// TIA Portal V19 export
DATA_BLOCK "RollformingMng"   // DB157
{ DB_Accessible_From_OPC_UA := 'FALSE' }
// stored: DBAccessibleFromOPCUA false, InstanceOfName RollformingMng_FB, InstanceOfType FB
"RollformingMng_FB"
   // VAR_INPUT
   //    AreaInterface : "AreaInterface";
   //    ZSI_Area : "udt_ZoneSafetyInterface";
   //    DataIn : Struct
   //       PbMaterialFwd : Bool;
   //       PbCutRest : Bool;
   //       PbCutWork : Bool;
   //       SensorMatPresence_Entry : Bool;
   //       SensorMatPresence_BeforeMW : Bool;
   //       SensorMatPresence_AfterMW : Bool;
   //       SensorMatPresence_ConveyorEntry : Bool;
   //    END_STRUCT;
   //    CIn : Struct
   //       PitTable : Struct
   //          IsAtRest : Bool;
   //          IsAtWork : Bool;
   //       END_STRUCT;
   //       Upstream : Struct
   //          EnableMove : Bool;
   //          InCycleOrEmptying : Bool;
   //          NextEndOfMaterial : Bool;
   //       END_STRUCT;
   //       PPrf : "PPrf_Data";
   //       ProdManager : "Prod_Part_Ctrl";
   //       Rollformer : Struct
   //          IsStandstill : Bool;
   //          InTargetPosition : Bool;
   //          TargetPosAx : LReal;
   //          ActualPosition : LReal;
   //          ActualVelocity : LReal;
   //       END_STRUCT;
   //       MwFakCalc : Struct
   //          ChangeRequest : Bool;
   //       END_STRUCT;
   //       FinalCut : Struct
   //          IsStandstill : Bool;
   //          AlarmsPresence : Bool;
   //          AllHeadAtRest : Bool;
   //          Avg_R_to_W_Time : Time;
   //          Avg_W_to_R_Time : Time;
   //          CutHead : Struct
   //             IsAtRest : Bool;
   //             IsAtWork : Bool;
   //          END_STRUCT;
   //          DrawHead : Struct
   //             IsAtRest : Bool;
   //             IsAtWork : Bool;
   //          END_STRUCT;
   //          MarkHead : Struct
   //             IsAtRest : Bool;
   //             IsAtWork : Bool;
   //          END_STRUCT;
   //       END_STRUCT;
   //       MaterialCounter : Struct
   //          AlrPresence : Bool;
   //          WngPresence : Bool;
   //          Data : "MatCountData";
   //       END_STRUCT;
   //       WeldReg : Struct
   //          ActTarget_P_ID : DInt;
   //          ActTarget_WeldPresence : Bool;
   //          ActTarget_WeldEndPos : LReal;
   //          NextTarget_P_ID : DInt;
   //          NextTarget_WeldPresence : Bool;
   //          NextTarget_WeldEndPos : LReal;
   //          WeldMIssingToFinalCut : LReal;
   //          WeldPresence : Bool;
   //       END_STRUCT;
   //       AccDecRollway : "udt_AccRollConveyor_COut_Manager";
   //    END_STRUCT;
   //    Config : Struct
   //       SensorsDelayOn : Time;
   //       SensorsDelayOff : Time;
   //       SensorExtractor_DelayOn : Time;
   //       SensorExtractor_DelayOff : Time;
   //    END_STRUCT;
   // END_VAR
   // VAR_OUTPUT
   //    MachineInterface : "MachineInterface";
   //    DataOut : Struct
   //       LampInPosition : Bool;
   //    END_STRUCT;
   //    COut : Struct
   //       PitTable : "ValveMachine_Manager";
   //       Rollformer : Struct
   //          Feed : "PositioningMachine_Manager";
   //       END_STRUCT;
   //       RegolazioneFormato : Struct
   //          LineSetup_Exe : Bool;
   //       END_STRUCT;
   //       ProdManager : Struct
   //          TargetDone : Bool;
   //          Heading : Bool;
   //          PartDone : "Prod_Part_Done";
   //       END_STRUCT;
   //       FlyingCarriage : "udt_FlyingCarriage_CIn";
   //       FinalCut : Struct
   //          CutHead : "ValveMachine_Manager";
   //          DrawHead : "ValveMachine_Manager";
   //          MarkHead : "ValveMachine_Manager";
   //          CutHead_Enable : Bool;
   //          DrawHead_Enable : Bool;
   //          MarkHead_Enable : Bool;
   //       END_STRUCT;
   //       AccRollConveyor : Struct
   //          Roll_FwdReq : Bool;
   //          PosCoda : LReal;
   //       END_STRUCT;
   //       FAK_UpdatePPrf : Struct
   //          FAK_Apply : Bool;
   //          FAK_Calculate : LReal;
   //       END_STRUCT;
   //       UpstreamLine : Struct
   //          LineVelocity : LReal;
   //       END_STRUCT;
   //       WeldReg : Struct
   //          ActTarget_P_ID : DInt;
   //          ActTarget_XStart : LReal;
   //          ActTarget_XEnd : LReal;
   //          NextTarget_P_ID : DInt;
   //          NextTarget_XStart : LReal;
   //          NextTarget_XEnd : LReal;
   //       END_STRUCT;
   //    END_STRUCT;
   // END_VAR
   // VAR_IN_OUT
   //    Pers : "udt_RollformingMng_Pers";
   // END_VAR
   // VAR
   //    Alarm : Struct
   //       MaterialMissing : Bool;
   //       MatCounterAlrPresence : Bool;
   //       NoTargetReady : Bool;
   //       ThreadingNotComplete : Bool;
   //       TooMuchNegativeMovRequired : Bool;
   //       PartCuttedManualTest : Bool;
   //       PartCuttedTooShort : Bool;
   //       DestinationLost : Bool;
   //       HeadingCutDone : Bool;
   //       STOP_Part_Recondition : Bool;
   //       STOP_Order_Complete : Bool;
   //       STOP_O_ACT_Empty : Bool;
   //       STOP_FineTurno : Bool;
   //       STOP_End_Of_Proroduction : Bool;
   //       STOP_ControlloQualita : Bool;
   //       STOP_Matrice_Colata_Coil : Bool;
   //    END_STRUCT;
   //    Warning : Struct
   //       NotAutReady : Bool;
   //       MatCounterWngPresence : Bool;
   //       RollformerLimitToPushMin : Bool;
   //       RollformerStopAwaitJobPerform : Bool;
   //       HeadingNotDone : Bool;
   //       StopInactivity : Bool;
   //       FlyingShear : Struct
   //          NotReachable : Bool;
   //          NotSynched : Bool;
   //          WorkByTimeout : Bool;
   //       END_STRUCT;
   //       SlowDownFromMes : Struct
   //          SLOW_Part_Recondition : Bool;
   //          SLOW_Order_Approach_To_Complete : Bool;
   //          SLOW_End_Of_Production : Bool;
   //       END_STRUCT;
   //       StopFromMes : Struct
   //          STOP_Part_Recondition : Bool;
   //          STOP_Order_Complete : Bool;
   //          STOP_O_ACT_Empty : Bool;
   //          STOP_End_Of_Proroduction : Bool;
   //          STOP_FineTurno : Bool;
   //          STOP_ControlloQualita : Bool;
   //          STOP_Matrice_Colata_Coil : Bool;
   //       END_STRUCT;
   //    END_STRUCT;
   //    HMI : Struct
   //       ProductionRateRequired : LReal;
   //       ProductionRateTargetReal : LReal;
   //       BufferCut : Struct
   //          Index : Int;
   //          ButtonDelete : Bool;
   //       END_STRUCT;
   //    END_STRUCT;
   //    Ctrl : Struct
   //       Stop_M1 : Bool;
   //       Stop_M2 : Bool;
   //       Stop : Bool;
   //       Rollformer : Struct
   //          SemiAut_PosAbs : Bool;
   //          SemiAut_Fwd : Bool;
   //          Aut_PosAbs : Bool;
   //          Aut_Fwd : Bool;
   //          Target_Vel : LReal;
   //          Target_Final : LReal;
   //          Target_Push : LReal;
   //          Target_Selected : LReal;
   //       END_STRUCT;
   //       FinalCut : Struct
   //          SemiAut_Rest : Bool;
   //          SemiAut_Work : Bool;
   //          Aut_Rest : Bool;
   //          Aut_Work : Bool;
   //       END_STRUCT;
   //    END_STRUCT;
   //    Sts : Struct
   //       IsStandstill : Bool;
   //       AlarmsPresence : Bool;
   //       WarningsPresence : Bool;
   //       Semiautomatic : Bool;
   //       SemiAut_Request : Bool;
   //       PbCutSemiAutoWork : Bool;
   //       LowSpeedPartsStart : Bool;
   //       FirstPartDone : Bool;
   //       ExtractionReq : Bool;
   //       CheckNewTarget : Bool;
   //       WeldSlowDown : Bool;
   //       MesSlowDown : Bool;
   //       Vel_FactorRateStep : LReal;
   //       Vel_Factor_New : LReal;
   //       StopInactivity : Bool;
   //       Rollformer : Struct
   //          IsStandstill : Bool;
   //          StopFeed : Struct
   //             Alarm : Bool;
   //             Safety : Bool;
   //             Cycle : Bool;
   //             Stations : Bool;
   //             Target : Bool;
   //             Presence : Bool;
   //             ProgramData : Bool;
   //             Upstream : Bool;
   //             Downstream : Bool;
   //             Limit : Bool;
   //             StillCutPerform : Bool;
   //          END_STRUCT;
   //          PosAbsEnable : Bool;
   //          FwdEnable : Bool;
   //          ExtraLow : Bool;
   //          PartsMissingToHighVel : Int;
   //          ActualTargetPosMatCountPos : LReal;
   //          Target_Valid : Bool;
   //          Target_Final_Valid : Bool;
   //          Target_Final_Reached : Bool;
   //          Target_Push_Valid : Bool;
   //          Target_Push_Reached : Bool;
   //          Target_SelectionCode : Int;
   //       END_STRUCT;
   //       Feeding : Struct
   //          StoppedForWork : Bool;
   //       END_STRUCT;
   //       FinalCut : Struct
   //          IsStandstill : Bool;
   //          WorkRequired : Bool;
   //          RestEnable : Bool;
   //          HeadingEnable : Bool;
   //          UseDrawHead : Bool;
   //          UseMarkHead : Bool;
   //          CutHead_WorkEnable : Bool;
   //          DrawHead_WorkEnable : Bool;
   //          MarkHead_WorkEnable : Bool;
   //       END_STRUCT;
   //    END_STRUCT;
   //    FlyingCutoff : "FlyingStation_Manager";
   //    CutLength : "CutLength";
   //    FeedLimit : "FeedLimiting";
   //    MatPresence_Entry1 : "DelayOnOff_R";
   //    MatPresence_Exit1 : "DelayOnOff_R";
   //    MatPresence_Exit2 : "DelayOnOff_R";
   //    MatPresence_Extr_IN : "DelayOnOff_R";
   //    MatPresence_Extr_OUT : "DelayOnOff_R";
   //    TON_Stop : TON_TIME;
   //    TOF_ProdRun : TOF_TIME;
   //    TON_NoTargetReady : TON_TIME;
   //    TON_StopInactivity : TON_TIME;
   //    AuxPE : Struct
   //       P_SemiAut_Request : Bool;
   //       P_PbCutRest : Bool;
   //       P_PbCutWork : Bool;
   //       P_SaveResult : Bool;
   //       N_FinalCut_AtRest1 : Bool;
   //       N_FinalCut_AtRest2 : Bool;
   //       P_FinalCut_AtWork : Bool;
   //    END_STRUCT;
   //    EmptyTarget : "udt_RollformingMng_Target";
   // END_VAR
BEGIN
END_DATA_BLOCK
